// TIA Portal V16 export
// export: Created 2023-05-12T08:05:31.8812854Z, ExportSetting WithDefaults, DisplayName Totally Integrated Automation Portal, DisplayVersion V16 Update 3, DisplayName TIA Portal Version Control Interface, DisplayVersion V16 Update 2, DisplayName TIA Portal Openness, DisplayVersion V16 Update 3, DisplayName SINAMICS Startdrive Advanced, DisplayVersion V16, DisplayName SINAMICS Startdrive G130, G150, S120, S150, SINAMICS MV, S210, DisplayVersion V16, DisplayName SINAMICS Startdrive G110M, G120, G120C, G120D, G120P, DisplayVersion V16, DisplayName STEP 7 Professional, DisplayVersion V16 Update 3, DisplayName STEP 7 Safety, DisplayVersion V16, DisplayName WinCC Advanced, DisplayVersion V16 Update 3
FUNCTION "CIP_ LINEA3" : Void   // FC55, STL
{ S7_Optimized_Access := 'FALSE' }
VERSION : 0.1
// stored: AutoNumber false, ParameterPassing false, UDAEnableTagReadback false
BEGIN

NETWORK
TITLE = PASO 1 PRIEMER ENJUEGE AGUA RECUPERADA
      A     "MARCAS CIP".MARCHA_CIP_LINEA_1;
      A(;
      O     "MARCAS CIP".SELECCION_CIP_AGUA_L1;
      O     "MARCAS CIP".SELECCION_CIP_CORTO_L1;
      O     "MARCAS CIP".SELECCION_CIP_LARGO_L1;
      );
      A     "MARCA_SELECCION_L3_CIP";
      AN    "PASOS CIP L3".paso_01_primer_enjuague;
      AN    "PASOS CIP L3".paso_02_vaciado_tanque;
      AN    "PASOS CIP L3".paso_03_preparacion_sosa;
      AN    "PASOS CIP L3".paso_04_enjuague_linea;
      AN    "PASOS CIP L3".paso_05_empuje_sosa;
      AN    "PASOS CIP L3".paso_06_sosa;
      AN    "PASOS CIP L3".paso_07_vaciado_tanque;
      AN    "PASOS CIP L3".paso_08_recuperar_sosa;
      AN    "PASOS CIP L3".paso_09_enjuague_sosa;
      AN    "PASOS CIP L3".paso_10_recup_enjuague;
      AN    "PASOS CIP L3".paso_11_vaciado_tanque;
      AN    "PASOS CIP L3".paso_12_preparar_acido;
      AN    "PASOS CIP L3".paso_13_enjuague_linea;
      AN    "PASOS CIP L3".paso_14_empuje_acido;
      AN    "PASOS CIP L3".paso_15_enjuague_linea;
      AN    "PASOS CIP L3".paso_16_vaciado_tanque;
      AN    "PASOS CIP L3".paso_17_recuperar_acido;
      AN    "PASOS CIP L3".paso_18_enjuague_acido;
      AN    "PASOS CIP L3".paso_19_recup_enjuague;

      AN    "PASOS CIP L3".paso_20_vaciado_tanque;

      AN    "PASOS CIP L3".paso_21;
      AN    "PASOS CIP L3".paso_22;
      AN    "PASOS CIP L3".paso_23;
      AN    "PASOS CIP L3".paso_24;
      S     "PASOS CIP L3".paso_01_primer_enjuague;

NETWORK
TITLE = PASO1: PRIMER ENJUAGUE
      A     "PASOS CIP L3".paso_01_primer_enjuague;
      A(;
      O     "MARCAS CIP".SELECCION_CIP_AGUA_L1;
      O     "MARCAS CIP".SELECCION_CIP_CORTO_L1;  // S5T#4M
      O     "MARCAS CIP".SELECCION_CIP_LARGO_L1;

      );
      A     "MARCAS CIP".MARCHA_CIP_LINEA_1;
      A     "MARCA_SELECCION_L3_CIP";
      L     "SP TIM L3 ESCALADO".TIM_PASO_1_L1;
      SD    "Tag_796";

NETWORK
TITLE = PASO 2: VACIADO TANQUE (SOLO BOMBA RETORNO CIP)
      A     "PASOS CIP L3".paso_01_primer_enjuague;
      A(;
      O     "MARCAS CIP".SELECCION_CIP_AGUA_L1;
      O     "MARCAS CIP".SELECCION_CIP_CORTO_L1;
      O     "MARCAS CIP".SELECCION_CIP_LARGO_L1;

      );
      A     "M_LIMPIEZA TANQUES_L1";
      A     "Tag_796";
      R     "PASOS CIP L3".paso_01_primer_enjuague;
      S     "PASOS CIP L3".paso_02_vaciado_tanque;

NETWORK
TITLE = 
      A     "PASOS CIP L3".paso_01_primer_enjuague;
      A(;
      O     "MARCAS CIP".SELECCION_CIP_CORTO_L1;
      O     "MARCAS CIP".SELECCION_CIP_LARGO_L1;
      );

      AN    "M_LIMPIEZA TANQUES_L1";
      A     "Tag_796";
      R     "PASOS CIP L3".paso_01_primer_enjuague;
      S     "PASOS CIP L3".paso_03_preparacion_sosa;

NETWORK
TITLE = 
      A     "PASOS CIP L3".paso_01_primer_enjuague;
      A     "MARCAS CIP".SELECCION_CIP_AGUA_L1;
      AN    "M_LIMPIEZA TANQUES_L1";
      A     "Tag_796";
      R     "PASOS CIP L3".paso_01_primer_enjuague;

      R     "MARCAS CIP".RUN_CIP_PASTE;
      R     "MARCAS CIP".RUN_CIP_L_LECHE_A_FLAN;
      R     "MARCAS CIP".RUN_CIP_L_LECHE_NATILLAS;

      R     "MARCAS CIP".MARCHA_CIP_LINEA_1;


NETWORK
TITLE = 
      A     "PASOS CIP L3".paso_02_vaciado_tanque;
      A(;
      O     "MARCAS CIP".SELECCION_CIP_AGUA_L1;
      O     "MARCAS CIP".SELECCION_CIP_CORTO_L1;
      O     "MARCAS CIP".SELECCION_CIP_LARGO_L1;
      );


      A     "MARCAS CIP".MARCHA_CIP_LINEA_1;
      A     "MARCA_SELECCION_L3_CIP";
      AN    "DETECTOR FLUJO RET_L2";
      L     S5T#30S;
      SD    "Tag_797";

NETWORK
TITLE = 
      A     "PASOS CIP L3".paso_02_vaciado_tanque;
      A(;
      O     "MARCAS CIP".SELECCION_CIP_CORTO_L1;
      O     "MARCAS CIP".SELECCION_CIP_LARGO_L1;
      );

      A     "Tag_797";
      AN    "DETECTOR FLUJO RET_L2";
      R     "PASOS CIP L3".paso_02_vaciado_tanque;
      S     "PASOS CIP L3".paso_03_preparacion_sosa;

NETWORK
TITLE = 
      A     "PASOS CIP L3".paso_02_vaciado_tanque;
      A     "MARCAS CIP".SELECCION_CIP_AGUA_L1;
      A     "Tag_797";
      AN    "DETECTOR FLUJO RET_L2";
      R     "PASOS CIP L3".paso_02_vaciado_tanque;

      R     "MARCAS CIP".RUN_CIP_PASTE;
      R     "MARCAS CIP".RUN_CIP_L_LECHE_A_FLAN;
      R     "MARCAS CIP".RUN_CIP_L_LECHE_NATILLAS;

      R     "MARCAS CIP".MARCHA_CIP_LINEA_1;


NETWORK
TITLE = PASO 3:PREPARACION SOSA
      A     "PASOS CIP L3".paso_03_preparacion_sosa;
      A(;
      O     "MARCAS CIP".SELECCION_CIP_CORTO_L1;
      O     "MARCAS CIP".SELECCION_CIP_LARGO_L1;
      );
      A     "MARCAS CIP".MARCHA_CIP_LINEA_1;
      A     "MARCA_SELECCION_L3_CIP";


      A     "TEMPERATURA SOSA".TEMPERATURA_OK_CAL;
      A     "CONDUCTIVIDAD_SOSA_L1".CONDUCTIVIDAD_OK;
      L     S5T#20S;
      SD    "Tag_798";

NETWORK
TITLE = 
      A     "PASOS CIP L3".paso_03_preparacion_sosa;
      A     "Tag_798";
      S     "PASOS CIP L3".paso_04_enjuague_linea;
      R     "PASOS CIP L3".paso_03_preparacion_sosa;


NETWORK
TITLE = PASO 4: ESPERA EMPUJE SOSA
      A     "PASOS CIP L3".paso_04_enjuague_linea;
      A(;
      O     "MARCAS CIP".SELECCION_CIP_CORTO_L1;
      O     "MARCAS CIP".SELECCION_CIP_LARGO_L1;
      );
      A     "MARCAS CIP".MARCHA_CIP_LINEA_1;
      A     "MARCA_SELECCION_L3_CIP";
      L     S5T#20S;
      SD    "Tag_799";

NETWORK
TITLE = 
      A     "PASOS CIP L3".paso_04_enjuague_linea;
      A     "Tag_799";
      R     "PASOS CIP L3".paso_04_enjuague_linea;
      S     "PASOS CIP L3".paso_05_empuje_sosa;


NETWORK
TITLE = PASO 5: EMPUJE SOSA
      A     "PASOS CIP L3".paso_05_empuje_sosa;
      A(;
      O     "MARCAS CIP".SELECCION_CIP_CORTO_L1;
      O     "MARCAS CIP".SELECCION_CIP_LARGO_L1;
      );
      A     "MARCAS CIP".MARCHA_CIP_LINEA_1;


      A     "MARCA_SELECCION_L3_CIP";
      A     "CONDUCT_RET_L2_SOSA".CONDUCTIVIDAD_OK;
      L     S5T#10S;
      SD    "Tag_800";

NETWORK
TITLE = 
      A     "PASOS CIP L3".paso_05_empuje_sosa;
      A     "Tag_800";
      A     "CONDUCT_RET_L2_SOSA".CONDUCTIVIDAD_OK;
      R     "PASOS CIP L3".paso_05_empuje_sosa;
      S     "PASOS CIP L3".paso_06_sosa;


NETWORK
TITLE = PASO 6: SOSA
      A     "PASOS CIP L3".paso_06_sosa;
      A(;
      O     "MARCAS CIP".SELECCION_CIP_CORTO_L1;
      O     "MARCAS CIP".SELECCION_CIP_LARGO_L1;  // S5T#10M
      );


      A     "MARCAS CIP".MARCHA_CIP_LINEA_1;
      A     "MARCA_SELECCION_L3_CIP";
      L     "SP TIM L3 ESCALADO".TIM_PASO_6_L1;
      SD    "Tag_801";

NETWORK
TITLE = 
      A     "PASOS CIP L3".paso_06_sosa;
      A(;
      O     "MARCAS CIP".SELECCION_CIP_CORTO_L1;
      O     "MARCAS CIP".SELECCION_CIP_LARGO_L1;
      );

      A     "Tag_801";
      A     "M_LIMPIEZA TANQUES_L1";
      R     "PASOS CIP L3".paso_06_sosa;
      S     "PASOS CIP L3".paso_07_vaciado_tanque;

NETWORK
TITLE = 
      A     "PASOS CIP L3".paso_06_sosa;
      A(;
      O     "MARCAS CIP".SELECCION_CIP_CORTO_L1;
      O     "MARCAS CIP".SELECCION_CIP_LARGO_L1;
      );
      A     "Tag_801";

      AN    "M_LIMPIEZA TANQUES_L1";
      A     "MARCA_SELECCION_L3_CIP";
      R     "PASOS CIP L3".paso_06_sosa;
      S     "PASOS CIP L3".paso_08_recuperar_sosa;

NETWORK
TITLE = PASO 7: VACIADO SI TANQUE
      A     "PASOS CIP L3".paso_07_vaciado_tanque;
      A(;
      O     "MARCAS CIP".SELECCION_CIP_CORTO_L1;
      O     "MARCAS CIP".SELECCION_CIP_LARGO_L1;
      );
      A     "MARCAS CIP".MARCHA_CIP_LINEA_1;


      A     "MARCA_SELECCION_L3_CIP";
      AN    "DETECTOR FLUJO RET_L2";
      L     S5T#30S;
      SD    "Tag_802";

NETWORK
TITLE = 
      A     "PASOS CIP L3".paso_07_vaciado_tanque;
      A     "Tag_802";
      A     "M_LIMPIEZA TANQUES_L1";
      R     "PASOS CIP L3".paso_07_vaciado_tanque;
      S     "PASOS CIP L3".paso_08_recuperar_sosa;


NETWORK
TITLE = PASO 8: RECUPERACION SOSA
      A     "PASOS CIP L3".paso_08_recuperar_sosa;
      A(;
      O     "MARCAS CIP".SELECCION_CIP_CORTO_L1;
      O     "MARCAS CIP".SELECCION_CIP_LARGO_L1;
      );
      A     "MARCAS CIP".MARCHA_CIP_LINEA_1;


      A     "MARCA_SELECCION_L3_CIP";
      AN    "CONDUCT_RET_L2_SOSA".CONDUCTIVIDAD_OK;
      L     S5T#10S;
      SD    "Tag_803";

NETWORK
TITLE = 
      A     "PASOS CIP L3".paso_08_recuperar_sosa;
      A     "Tag_803";
      AN    "CONDUCT_RET_L2_SOSA".CONDUCTIVIDAD_OK;
      R     "PASOS CIP L3".paso_08_recuperar_sosa;
      S     "PASOS CIP L3".paso_09_enjuague_sosa;


NETWORK
TITLE = PASO 9: ENJUAGUE SOSA
      A     "PASOS CIP L3".paso_09_enjuague_sosa;
      A(;
      O     "MARCAS CIP".SELECCION_CIP_CORTO_L1;
      O     "MARCAS CIP".SELECCION_CIP_LARGO_L1;
      );
      A     "MARCAS CIP".MARCHA_CIP_LINEA_1;
      A     "MARCA_SELECCION_L3_CIP";
//      UN    "CONDUCT_RET_L1_AGUA".CONDUCTIVIDAD_OK
//      L     S5T#1M40S
      L     "SP TIM L3 ESCALADO".TIM_PASO_9_L1;
      SD    "Tag_804";

NETWORK
TITLE = 
      A     "PASOS CIP L3".paso_09_enjuague_sosa;
      A     "Tag_804";
      R     "PASOS CIP L3".paso_09_enjuague_sosa;
      S     "PASOS CIP L3".paso_10_recup_enjuague;


NETWORK
TITLE = PASO10:RECUPERACION ENJUAGUE SOSA
      A     "PASOS CIP L3".paso_10_recup_enjuague;
      A(;
      O     "MARCAS CIP".SELECCION_CIP_CORTO_L1;
      O     "MARCAS CIP".SELECCION_CIP_LARGO_L1;
      );


      A     "MARCAS CIP".MARCHA_CIP_LINEA_1;
      A     "MARCA_SELECCION_L3_CIP";
      L     "SP TIM L3 ESCALADO".TIM_PASO_10_L1;
      SD    "Tag_805";

NETWORK
TITLE = 
      A     "PASOS CIP L3".paso_10_recup_enjuague;
      A     "Tag_805";
      A     "M_LIMPIEZA TANQUES_L1";
      R     "PASOS CIP L3".paso_10_recup_enjuague;
      S     "PASOS CIP L3".paso_11_vaciado_tanque;


NETWORK
TITLE = 
      A     "PASOS CIP L3".paso_10_recup_enjuague;
      A     "MARCAS CIP".SELECCION_CIP_LARGO_L1;
      A     "Tag_805";
      AN    "M_LIMPIEZA TANQUES_L1";
      R     "PASOS CIP L3".paso_10_recup_enjuague;

      S     "PASOS CIP L3".paso_12_preparar_acido;

NETWORK
TITLE = 
      A     "PASOS CIP L3".paso_10_recup_enjuague;
      A     "MARCAS CIP".SELECCION_CIP_CORTO_L1;
      A     "Tag_805";
      AN    "M_LIMPIEZA TANQUES_L1";
      R     "PASOS CIP L3".paso_10_recup_enjuague;

      R     "MARCAS CIP".RUN_CIP_PASTE;
      R     "MARCAS CIP".RUN_CIP_L_LECHE_A_FLAN;
      R     "MARCAS CIP".RUN_CIP_L_LECHE_NATILLAS;

      R     "MARCAS CIP".MARCHA_CIP_LINEA_1;


NETWORK
TITLE = PASO 11: VACIADO SI TANQUE
      A     "PASOS CIP L3".paso_11_vaciado_tanque;
      A(;
      O     "MARCAS CIP".SELECCION_CIP_CORTO_L1;
      O     "MARCAS CIP".SELECCION_CIP_LARGO_L1;
      );
      A     "MARCAS CIP".MARCHA_CIP_LINEA_1;


      A     "MARCA_SELECCION_L3_CIP";
      AN    "DETECTOR FLUJO RET_L2";
      L     S5T#30S;
      SD    "Tag_806";

NETWORK
TITLE = 
      A     "PASOS CIP L3".paso_11_vaciado_tanque;
      A     "MARCAS CIP".SELECCION_CIP_LARGO_L1;
      A     "Tag_806";
      AN    "DETECTOR FLUJO RET_L2";
      R     "PASOS CIP L3".paso_11_vaciado_tanque;

      S     "PASOS CIP L3".paso_12_preparar_acido;

NETWORK
TITLE = 
      A     "PASOS CIP L3".paso_11_vaciado_tanque;
      A     "MARCAS CIP".SELECCION_CIP_CORTO_L1;
      A     "Tag_806";
      AN    "DETECTOR FLUJO RET_L2";
      R     "PASOS CIP L3".paso_11_vaciado_tanque;

      R     "MARCAS CIP".RUN_CIP_PASTE;
      R     "MARCAS CIP".RUN_CIP_L_LECHE_A_FLAN;
      R     "MARCAS CIP".RUN_CIP_L_LECHE_NATILLAS;

      R     "MARCAS CIP".MARCHA_CIP_LINEA_1;


NETWORK
TITLE = PASO 12: PREPARACION ACIDO
      A     "PASOS CIP L3".paso_12_preparar_acido;
      A     "MARCAS CIP".SELECCION_CIP_LARGO_L1;
      A     "MARCAS CIP".MARCHA_CIP_LINEA_1;
      A     "MARCA_SELECCION_L3_CIP";
      A     "TEMPERATURA ACIDO".TEMPERATURA_OK_CAL;
      A     "CONDUCTIVIDAD_ACIDO_L1".CONDUCTIVIDAD_OK;
      L     S5T#20S;
      SD    "Tag_807";

NETWORK
TITLE = 
      A     "PASOS CIP L3".paso_12_preparar_acido;
      A     "Tag_807";
      R     "PASOS CIP L3".paso_12_preparar_acido;
      S     "PASOS CIP L3".paso_13_enjuague_linea;


NETWORK
TITLE = PASO 13:ESPERA EMPUJE ACIDO
      A     "PASOS CIP L3".paso_13_enjuague_linea;
      A     "MARCAS CIP".SELECCION_CIP_LARGO_L1;
      A     "MARCAS CIP".MARCHA_CIP_LINEA_1;
      A     "MARCA_SELECCION_L3_CIP";
      L     S5T#20S;
      SD    "Tag_808";

NETWORK
TITLE = 
      A     "PASOS CIP L3".paso_13_enjuague_linea;
      A     "Tag_808";
      R     "PASOS CIP L3".paso_13_enjuague_linea;
      S     "PASOS CIP L3".paso_14_empuje_acido;


NETWORK
TITLE = PASO 14: EMPUJE ACIDO
      A     "PASOS CIP L3".paso_14_empuje_acido;
      A     "MARCAS CIP".SELECCION_CIP_LARGO_L1;
      A     "MARCAS CIP".MARCHA_CIP_LINEA_1;
      A     "MARCA_SELECCION_L3_CIP";
      A     "CONDUCT_RET_L2_ACIDO".CONDUCTIVIDAD_OK;
      L     S5T#10S;


      SD    "Tag_809";

NETWORK
TITLE = 
      A     "PASOS CIP L3".paso_14_empuje_acido;
      A     "Tag_809";
      R     "PASOS CIP L3".paso_14_empuje_acido;
      S     "PASOS CIP L3".paso_15_enjuague_linea;


NETWORK
TITLE = PASO 15:ACIDO
      A     "PASOS CIP L3".paso_15_enjuague_linea;
      A     "MARCAS CIP".SELECCION_CIP_LARGO_L1;
      A     "MARCAS CIP".MARCHA_CIP_LINEA_1;
      A     "MARCA_SELECCION_L3_CIP";  //  S5T#10M
      L     "SP TIM L3 ESCALADO".TIM_PASO_15_L1;


      SD    "Tag_810";

NETWORK
TITLE = Variable provisional
      A     "PASOS CIP L3".paso_15_enjuague_linea;
      A     "Tag_810";
      A     "M_LIMPIEZA TANQUES_L1";
      R     "PASOS CIP L3".paso_15_enjuague_linea;
      S     "PASOS CIP L3".paso_16_vaciado_tanque;


NETWORK
TITLE = Variable provisional
      A     "PASOS CIP L3".paso_15_enjuague_linea;
      A     "Tag_810";
      AN    "M_LIMPIEZA TANQUES_L1";
      R     "PASOS CIP L3".paso_15_enjuague_linea;
      S     "PASOS CIP L3".paso_17_recuperar_acido;


NETWORK
TITLE = PASO 16: VACIADO SI TANQUES
      A     "PASOS CIP L3".paso_16_vaciado_tanque;
      A     "MARCAS CIP".SELECCION_CIP_LARGO_L1;
      A     "MARCAS CIP".MARCHA_CIP_LINEA_1;
      A     "MARCA_SELECCION_L3_CIP";
      AN    "DETECTOR FLUJO RET_L2";
      L     S5T#30S;


      SD    "Tag_811";

NETWORK
TITLE = Variable provisional
      A     "PASOS CIP L3".paso_16_vaciado_tanque;
      A     "Tag_811";
      AN    "DETECTOR FLUJO RET_L2";
      R     "PASOS CIP L3".paso_16_vaciado_tanque;
      S     "PASOS CIP L3".paso_17_recuperar_acido;


NETWORK
TITLE = PASO 17: RECUPERACION ACIDO
      A     "PASOS CIP L3".paso_17_recuperar_acido;
      A     "MARCAS CIP".SELECCION_CIP_LARGO_L1;
      A     "MARCAS CIP".MARCHA_CIP_LINEA_1;
      A     "MARCA_SELECCION_L3_CIP";
      AN    "CONDUCT_RET_L2_ACIDO".CONDUCTIVIDAD_OK;
      L     S5T#10S;
      SD    "Tag_812";

NETWORK
TITLE = Variable provisional
      A     "PASOS CIP L3".paso_17_recuperar_acido;
      A     "Tag_812";
      AN    "CONDUCT_RET_L2_ACIDO".CONDUCTIVIDAD_OK;
      R     "PASOS CIP L3".paso_17_recuperar_acido;
      S     "PASOS CIP L3".paso_18_enjuague_acido;


NETWORK
TITLE = PASO 18: ENJUAGUE ACIDO
      A     "PASOS CIP L3".paso_18_enjuague_acido;
      A     "MARCAS CIP".SELECCION_CIP_LARGO_L1;
      A     "MARCAS CIP".MARCHA_CIP_LINEA_1;
      A     "MARCA_SELECCION_L3_CIP";
//      UN    "CONDUCT_RET_L1_AGUA".CONDUCTIVIDAD_OK
//      L     S5T#1M40S
      L     "SP TIM L3 ESCALADO".TIM_PASO_18_L1;
      SD    "Tag_813";

NETWORK
TITLE = 
      A     "PASOS CIP L3".paso_18_enjuague_acido;
      A     "Tag_813";
      R     "PASOS CIP L3".paso_18_enjuague_acido;
      S     "PASOS CIP L3".paso_19_recup_enjuague;


NETWORK
TITLE = PASO 19:RECUPERACION ENJUAGUE ACIDO
      A     "PASOS CIP L3".paso_19_recup_enjuague;
      A     "MARCAS CIP".SELECCION_CIP_LARGO_L1;
      A     "MARCAS CIP".MARCHA_CIP_LINEA_1;
      A     "MARCA_SELECCION_L3_CIP";  // S5T#2M
      L     "SP TIM L3 ESCALADO".TIM_PASO_19_L1;


      SD    "Tag_814";

NETWORK
TITLE = 
      A     "PASOS CIP L3".paso_19_recup_enjuague;
      A     "M_LIMPIEZA TANQUES_L1";
      A     "Tag_814";
      R     "PASOS CIP L3".paso_19_recup_enjuague;
      S     "PASOS CIP L3".paso_20_vaciado_tanque;


NETWORK
TITLE = 
      A     "PASOS CIP L3".paso_19_recup_enjuague;
      AN    "M_LIMPIEZA TANQUES_L1";
      A     "Tag_814";
      R     "PASOS CIP L3".paso_19_recup_enjuague;

      R     "MARCAS CIP".RUN_CIP_PASTE;
      R     "MARCAS CIP".RUN_CIP_L_LECHE_A_FLAN;
      R     "MARCAS CIP".RUN_CIP_L_LECHE_NATILLAS;

      R     "MARCAS CIP".MARCHA_CIP_LINEA_1;


NETWORK
TITLE = PASO 19: VACIADO SI TANQUES
      A     "PASOS CIP L3".paso_20_vaciado_tanque;
      A     "MARCAS CIP".SELECCION_CIP_LARGO_L1;
      A     "MARCAS CIP".MARCHA_CIP_LINEA_1;
      A     "MARCA_SELECCION_L3_CIP";
      AN    "DETECTOR FLUJO RET_L2";
      L     S5T#50S;


      SD    "Tag_815";

NETWORK
TITLE = FIN DE CICLO
      A     "PASOS CIP L3".paso_20_vaciado_tanque;
      A     "Tag_815";
      R     "PASOS CIP L3".paso_20_vaciado_tanque;


      R     "MARCAS CIP".RUN_CIP_PASTE;
      R     "MARCAS CIP".RUN_CIP_L_LECHE_A_FLAN;
      R     "MARCAS CIP".RUN_CIP_L_LECHE_NATILLAS;

      R     "MARCAS CIP".MARCHA_CIP_LINEA_1;




NETWORK
TITLE = Variable prvisional

      AN    "MARCAS CIP".MARCHA_CIP_LINEA_1;


      R     "PASOS CIP L3".paso_01_primer_enjuague;
      R     "PASOS CIP L3".paso_02_vaciado_tanque;
      R     "PASOS CIP L3".paso_03_preparacion_sosa;
      R     "PASOS CIP L3".paso_04_enjuague_linea;
      R     "PASOS CIP L3".paso_05_empuje_sosa;
      R     "PASOS CIP L3".paso_06_sosa;
      R     "PASOS CIP L3".paso_07_vaciado_tanque;
      R     "PASOS CIP L3".paso_08_recuperar_sosa;
      R     "PASOS CIP L3".paso_09_enjuague_sosa;
      R     "PASOS CIP L3".paso_10_recup_enjuague;
      R     "PASOS CIP L3".paso_11_vaciado_tanque;
      R     "PASOS CIP L3".paso_12_preparar_acido;
      R     "PASOS CIP L3".paso_13_enjuague_linea;
      R     "PASOS CIP L3".paso_14_empuje_acido;
      R     "PASOS CIP L3".paso_15_enjuague_linea;
      R     "PASOS CIP L3".paso_16_vaciado_tanque;
      R     "PASOS CIP L3".paso_17_recuperar_acido;
      R     "PASOS CIP L3".paso_18_enjuague_acido;
      R     "PASOS CIP L3".paso_19_recup_enjuague;
      R     "PASOS CIP L3".paso_20_vaciado_tanque;







END_FUNCTION
